// TIA Portal V20 export
TYPE "typeEm7MonitoringCmStatus"
// stored: Access Published, Namespace Unit1
   STRUCT
      ngKickerAxis { ExternalWritable := 'False'} : "LBC_typeAxisControlNodeMonitoring";
      passKickerAxis { ExternalWritable := 'False'} : "LBC_typeAxisControlNodeMonitoring";
      cutConvAxis { ExternalWritable := 'False'} : "LBC_typeAxisControlNodeMonitoring";
      ngConvAxis { ExternalWritable := 'False'} : "LBC_typeAxisControlNodeMonitoring";
      stack1ConvAxis { ExternalWritable := 'False'} : "LBC_typeAxisControlNodeMonitoring";
      stack2ConvAxis { ExternalWritable := 'False'} : "LBC_typeAxisControlNodeMonitoring";
      convVirtualAxis { ExternalWritable := 'False'} : "LBC_typeAxisControlNodeMonitoring";
      cutConvRingBlow { ExternalWritable := 'False'} : "LBC_typeSinaSpeedControlNodeMonitoring";
      ngConvRingBlow { ExternalWritable := 'False'} : "LBC_typeSinaSpeedControlNodeMonitoring";
      stack2ConvRingBlow { ExternalWritable := 'False'} : "LBC_typeSinaSpeedControlNodeMonitoring";
      ngBoxLockCyl { ExternalWritable := 'False'} : "LBC_typeTwoWayActuatorControlNodeMonitoring";
      ngBoxDetect { ExternalWritable := 'False'} : "LBC_typeDigitalSignalControlNodeMonitoring";
      ngBoxFull { ExternalWritable := 'False'} : "LBC_typeDigitalSignalControlNodeMonitoring";
      ngKickerDetect { ExternalWritable := 'False'} : "LBC_typeDigitalSignalControlNodeMonitoring";
      passKickerDetect { ExternalWritable := 'False'} : "LBC_typeDigitalSignalControlNodeMonitoring";
      stack1ConvElecDetect { ExternalWritable := 'False'} : "LBC_typeDigitalSignalControlNodeMonitoring";
      stack2ConvElecDetect { ExternalWritable := 'False'} : "LBC_typeDigitalSignalControlNodeMonitoring";
   END_STRUCT;
END_TYPE
